{attribute 'TcDependOnClassFactory' := 'Welding_Control_Circle_86s'}
FUNCTION_BLOCK FB_Welding_Control_Circle_86s EXTENDS FB_TcMatSimObject
VAR_INPUT
	stInput: ST_Welding_Control_Circle_86s_Input;
END_VAR
VAR_OUTPUT
	stOutput: ST_Welding_Control_Circle_86s_Output;
END_VAR
VAR
	stInitData: ST_Welding_Control_Circle_86s_InitData;
	arrDataAreas: ARRAY[1..2] OF ST_TcMatSimObjectDataAreaInfo;
	bParametersVerified: BOOL;
END_VAR

PROPERTY CallBy_Online : TctModuleCallByType
GET
hResult := GetObjPara(16#00000000,sizeof(CallBy_Online),adr(CallBy_Online));
END_GET
SET
hResult := SetObjPara(16#00000000,sizeof(CallBy_Online),adr(CallBy_Online));
END_SET
END_PROPERTY

PROPERTY CallBy_Startup : TctModuleCallByType
GET
CallBy_Startup := stInitData.CallBy;
END_GET
SET
stInitData.CallBy := CallBy_Startup;
END_SET
END_PROPERTY

PROPERTY ContextInfoArr_0_TaskCycleTimeNs_Online : UDINT
GET
hResult := GetObjPara(16#03002080,sizeof(ContextInfoArr_0_TaskCycleTimeNs_Online),adr(ContextInfoArr_0_TaskCycleTimeNs_Online));
END_GET
SET
hResult := SetObjPara(16#03002080,sizeof(ContextInfoArr_0_TaskCycleTimeNs_Online),adr(ContextInfoArr_0_TaskCycleTimeNs_Online));
END_SET
END_PROPERTY

PROPERTY ContextInfoArr_0_TaskCycleTimeNs_Startup : UDINT
GET
ContextInfoArr_0_TaskCycleTimeNs_Startup := stInitData.ContextInfoArr_0_TaskCycleTimeNs;
END_GET
SET
stInitData.ContextInfoArr_0_TaskCycleTimeNs := ContextInfoArr_0_TaskCycleTimeNs_Startup;
END_SET
END_PROPERTY

PROPERTY ContextInfoArr_0_TaskOid_Online : OTCID
GET
hResult := GetObjPara(16#03002060,sizeof(ContextInfoArr_0_TaskOid_Online),adr(ContextInfoArr_0_TaskOid_Online));
END_GET
SET
hResult := SetObjPara(16#03002060,sizeof(ContextInfoArr_0_TaskOid_Online),adr(ContextInfoArr_0_TaskOid_Online));
END_SET
END_PROPERTY

PROPERTY ContextInfoArr_0_TaskOid_Startup : OTCID
GET
ContextInfoArr_0_TaskOid_Startup := stInitData.ContextInfoArr_0_TaskOid;
END_GET
SET
stInitData.ContextInfoArr_0_TaskOid := ContextInfoArr_0_TaskOid_Startup;
END_SET
END_PROPERTY

PROPERTY ContextInfoArr_0_TaskPort_Online : UINT
GET
hResult := GetObjPara(16#03002090,sizeof(ContextInfoArr_0_TaskPort_Online),adr(ContextInfoArr_0_TaskPort_Online));
END_GET
SET
hResult := SetObjPara(16#03002090,sizeof(ContextInfoArr_0_TaskPort_Online),adr(ContextInfoArr_0_TaskPort_Online));
END_SET
END_PROPERTY

PROPERTY ContextInfoArr_0_TaskPort_Startup : UINT
GET
ContextInfoArr_0_TaskPort_Startup := stInitData.ContextInfoArr_0_TaskPort;
END_GET
SET
stInitData.ContextInfoArr_0_TaskPort := ContextInfoArr_0_TaskPort_Startup;
END_SET
END_PROPERTY

PROPERTY ContextInfoArr_0_TaskPriority_Online : UDINT
GET
hResult := GetObjPara(16#03002070,sizeof(ContextInfoArr_0_TaskPriority_Online),adr(ContextInfoArr_0_TaskPriority_Online));
END_GET
SET
hResult := SetObjPara(16#03002070,sizeof(ContextInfoArr_0_TaskPriority_Online),adr(ContextInfoArr_0_TaskPriority_Online));
END_SET
END_PROPERTY

PROPERTY ContextInfoArr_0_TaskPriority_Startup : UDINT
GET
ContextInfoArr_0_TaskPriority_Startup := stInitData.ContextInfoArr_0_TaskPriority;
END_GET
SET
stInitData.ContextInfoArr_0_TaskPriority := ContextInfoArr_0_TaskPriority_Startup;
END_SET
END_PROPERTY

PROPERTY ContextInfoArr_0_TaskSortOrder_Online : UDINT
GET
hResult := GetObjPara(16#030020b0,sizeof(ContextInfoArr_0_TaskSortOrder_Online),adr(ContextInfoArr_0_TaskSortOrder_Online));
END_GET
SET
hResult := SetObjPara(16#030020b0,sizeof(ContextInfoArr_0_TaskSortOrder_Online),adr(ContextInfoArr_0_TaskSortOrder_Online));
END_SET
END_PROPERTY

PROPERTY ContextInfoArr_0_TaskSortOrder_Startup : UDINT
GET
ContextInfoArr_0_TaskSortOrder_Startup := stInitData.ContextInfoArr_0_TaskSortOrder;
END_GET
SET
stInitData.ContextInfoArr_0_TaskSortOrder := ContextInfoArr_0_TaskSortOrder_Startup;
END_SET
END_PROPERTY

PROPERTY CycleUpdateExecuted_Online : BOOL
GET
hResult := GetObjPara(16#00000004,sizeof(CycleUpdateExecuted_Online),adr(CycleUpdateExecuted_Online));
END_GET
SET
hResult := SetObjPara(16#00000004,sizeof(CycleUpdateExecuted_Online),adr(CycleUpdateExecuted_Online));
END_SET
END_PROPERTY

METHOD Execute : HRESULT

IF (SUCCEEDED(hResult)) THEN
  hResult := VerifyParameters();
END_IF

	// update DataArea information
SetDataAreaInfo(ADR(arrDataAreas),2);
	
	// call base method
Execute := SUPER^.Execute();
END_METHOD

PROPERTY ExecuteModelCode_Online : BOOL
GET
hResult := GetObjPara(16#00000008,sizeof(ExecuteModelCode_Online),adr(ExecuteModelCode_Online));
END_GET
SET
hResult := SetObjPara(16#00000008,sizeof(ExecuteModelCode_Online),adr(ExecuteModelCode_Online));
END_SET
END_PROPERTY

PROPERTY ExecuteModelCode_Startup : BOOL
GET
ExecuteModelCode_Startup := stInitData.ExecuteModelCode;
END_GET
SET
stInitData.ExecuteModelCode := ExecuteModelCode_Startup;
END_SET
END_PROPERTY

PROPERTY ExecutionSequence_Online : TctModuleExecutionSequenceType
GET
hResult := GetObjPara(16#00000001,sizeof(ExecutionSequence_Online),adr(ExecutionSequence_Online));
END_GET
SET
hResult := SetObjPara(16#00000001,sizeof(ExecutionSequence_Online),adr(ExecutionSequence_Online));
END_SET
END_PROPERTY

PROPERTY ExecutionSequence_Startup : TctModuleExecutionSequenceType
GET
ExecutionSequence_Startup := stInitData.ExecutionSequence;
END_GET
SET
stInitData.ExecutionSequence := ExecutionSequence_Startup;
END_SET
END_PROPERTY

METHOD FB_init : BOOL
VAR_INPUT
	/// if TRUE, the retain variables are initialized (warm start / cold start)
	bInitRetains: BOOL;
	/// if TRUE, the instance afterwards gets moved into the copy code (online change)
	bInCopyCode: BOOL;
	oid: OTCID;
END_VAR
VAR
	clsId: CLSID;
END_VAR

// initialize flags
bParametersVerified := false;
                    
// set module class id for compatibility check
clsId.Data1 := 16#4f7c9520;
clsId.Data2 := 16#5e7b;
clsId.Data3 := 16#4579;
clsId.Data4[0] := 16#be;
clsId.Data4[1] := 16#6e;
clsId.Data4[2] := 16#10;
clsId.Data4[3] := 16#c0;
clsId.Data4[4] := 16#eb;
clsId.Data4[5] := 16#37;
clsId.Data4[6] := 16#31;
clsId.Data4[7] := 16#6d;

AssignClassId(clsId);
                    
// initialize InitData structure with default values              
stInitData.CallByHdr.indexGroup := 0;
stInitData.CallByHdr.indexOffset := 16#00000000;
stInitData.CallByHdr.cbData := SIZEOF(stInitData.CallBy);
stInitData.CallBy := TctModuleCallByType.Module;
stInitData.ExecutionSequenceHdr.indexGroup := 0;
stInitData.ExecutionSequenceHdr.indexOffset := 16#00000001;
stInitData.ExecutionSequenceHdr.cbData := SIZEOF(stInitData.ExecutionSequence);
stInitData.ExecutionSequence := TctModuleExecutionSequenceType.StateUpdateAfterOutputMapping;
stInitData.StepSizeHdr.indexGroup := 0;
stInitData.StepSizeHdr.indexOffset := 16#00000002;
stInitData.StepSizeHdr.cbData := SIZEOF(stInitData.StepSize);
stInitData.StepSize := TctStepSizeType.UseTaskCycleTime;
stInitData.ExecuteModelCodeHdr.indexGroup := 0;
stInitData.ExecuteModelCodeHdr.indexOffset := 16#00000008;
stInitData.ExecuteModelCodeHdr.cbData := SIZEOF(stInitData.ExecuteModelCode);
stInitData.ExecuteModelCode := 1;
stInitData.ContextInfoArr_0_TaskOidHdr.indexGroup := 0;
stInitData.ContextInfoArr_0_TaskOidHdr.indexOffset := 16#03002060;
stInitData.ContextInfoArr_0_TaskOidHdr.cbData := SIZEOF(stInitData.ContextInfoArr_0_TaskOid);
stInitData.ContextInfoArr_0_TaskPriorityHdr.indexGroup := 0;
stInitData.ContextInfoArr_0_TaskPriorityHdr.indexOffset := 16#03002070;
stInitData.ContextInfoArr_0_TaskPriorityHdr.cbData := SIZEOF(stInitData.ContextInfoArr_0_TaskPriority);
stInitData.ContextInfoArr_0_TaskCycleTimeNsHdr.indexGroup := 0;
stInitData.ContextInfoArr_0_TaskCycleTimeNsHdr.indexOffset := 16#03002080;
stInitData.ContextInfoArr_0_TaskCycleTimeNsHdr.cbData := SIZEOF(stInitData.ContextInfoArr_0_TaskCycleTimeNs);
stInitData.ContextInfoArr_0_TaskPortHdr.indexGroup := 0;
stInitData.ContextInfoArr_0_TaskPortHdr.indexOffset := 16#03002090;
stInitData.ContextInfoArr_0_TaskPortHdr.cbData := SIZEOF(stInitData.ContextInfoArr_0_TaskPort);
stInitData.ContextInfoArr_0_TaskSortOrderHdr.indexGroup := 0;
stInitData.ContextInfoArr_0_TaskSortOrderHdr.indexOffset := 16#030020b0;
stInitData.ContextInfoArr_0_TaskSortOrderHdr.cbData := SIZEOF(stInitData.ContextInfoArr_0_TaskSortOrder);
stInitData.Header.cbData := SIZEOF(stInitData)-SIZEOF(stInitData.Header);
stInitData.Header.uiElmCnt := 9;


// set pointer to InitData structure
SetInitDataInfo(ADR(stInitData));

// set DataArea information
SetDataAreaInfo(ADR(arrDataAreas),2);
arrDataAreas[1].nDataAreaId := 0;
arrDataAreas[1].nSize := SIZEOF(stInput);
arrDataAreas[1].pPlcVar := ADR(stInput);
arrDataAreas[1].pModuleProcImg := 0;
arrDataAreas[1].eDataAreaType := E_TcMatSimDataAreaType.InputDst;
arrDataAreas[2].nDataAreaId := 1;
arrDataAreas[2].nSize := SIZEOF(stOutput);
arrDataAreas[2].pPlcVar := ADR(stOutput);
arrDataAreas[2].pModuleProcImg := 0;
arrDataAreas[2].eDataAreaType := E_TcMatSimDataAreaType.OutputSrc;


// initialize basic interface pointers and return
FB_init := SUCCEEDED(Init(oid));
END_METHOD

PROPERTY InitData : ST_Welding_Control_Circle_86s_InitData
GET
InitData := stInitData;
END_GET
SET
stInitData := InitData;
END_SET
END_PROPERTY

PROPERTY Input_Online : ExtU_output_WeldingDiameter10_T
GET
hResult := GetObjPara(16#80000000,sizeof(Input_Online),adr(Input_Online));
END_GET
SET
hResult := SetObjPara(16#80000000,sizeof(Input_Online),adr(Input_Online));
END_SET
END_PROPERTY

{attribute 'object_name' := 'Internal_SetObjState'}
METHOD PROTECTED Internal_SetObjState
VAR_INPUT
	hr: REFERENCE TO HRESULT;
	nextState: TCOM_STATE;
END_VAR

// update pointer to InitData structure
SetInitDataInfo(ADR(stInitData));
// call base method
SUPER^.Internal_SetObjState(hr,nextState);
END_METHOD

PROPERTY MdlInitialized_Online : BOOL
GET
hResult := GetObjPara(16#00000003,sizeof(MdlInitialized_Online),adr(MdlInitialized_Online));
END_GET
SET
hResult := SetObjPara(16#00000003,sizeof(MdlInitialized_Online),adr(MdlInitialized_Online));
END_SET
END_PROPERTY

PROPERTY ModuleBuildInfo_Online : TctModuleBuildInfoType
GET
hResult := GetObjPara(16#00000007,sizeof(ModuleBuildInfo_Online),adr(ModuleBuildInfo_Online));
END_GET
SET
hResult := SetObjPara(16#00000007,sizeof(ModuleBuildInfo_Online),adr(ModuleBuildInfo_Online));
END_SET
END_PROPERTY

PROPERTY ModuleInfo_Online : TctModuleInfoType
GET
hResult := GetObjPara(16#00000006,sizeof(ModuleInfo_Online),adr(ModuleInfo_Online));
END_GET
SET
hResult := SetObjPara(16#00000006,sizeof(ModuleInfo_Online),adr(ModuleInfo_Online));
END_SET
END_PROPERTY

{attribute 'object_name' := 'SaveOnlineParametersForInit'}
METHOD SaveOnlineParametersForInit : HRESULT
VAR
	idx: UINT;
	pInitElemHdr: POINTER TO TComInitDataElmHdr;
	pData: PVOID;
	nData: UDINT;
END_VAR
VAR CONSTANT
	nInitDataAlignment: UDINT := 4;
END_VAR

// update pointer to InitData structure
SetInitDataInfo(ADR(stInitData));
// call base method
SaveOnlineParametersForInit := SUPER^.SaveOnlineParametersForInit();
END_METHOD

PROPERTY SimulinkTime_Online : LREAL
GET
hResult := GetObjPara(16#00000005,sizeof(SimulinkTime_Online),adr(SimulinkTime_Online));
END_GET
SET
hResult := SetObjPara(16#00000005,sizeof(SimulinkTime_Online),adr(SimulinkTime_Online));
END_SET
END_PROPERTY

PROPERTY StepSize_Online : TctStepSizeType
GET
hResult := GetObjPara(16#00000002,sizeof(StepSize_Online),adr(StepSize_Online));
END_GET
SET
hResult := SetObjPara(16#00000002,sizeof(StepSize_Online),adr(StepSize_Online));
END_SET
END_PROPERTY

PROPERTY StepSize_Startup : TctStepSizeType
GET
StepSize_Startup := stInitData.StepSize;
END_GET
SET
stInitData.StepSize := StepSize_Startup;
END_SET
END_PROPERTY

{attribute 'object_name' := 'VerifyParameters'}
METHOD PRIVATE VerifyParameters : HRESULT
VAR
	moduleCallByParam: TctModuleCallByType;
END_VAR

IF (bParametersVerified) THEN
  VerifyParameters := Tc2_System.E_HRESULTAdsErr.HRESULT_ADS_NOERROR;
ELSE
  VerifyParameters := GetObjPara(stInitData.CallByHdr.indexOffset,SIZEOF(moduleCallByParam),ADR(moduleCallByParam));
  
  // check the "CallBy" parameter to be set to "Module"
  IF (SUCCEEDED(VerifyParameters) AND (moduleCallByParam <> TctModuleCallByType.Module)) THEN
      VerifyParameters := Tc2_System.E_HRESULTAdsErr.INVALIDPARM;
  END_IF
  
  // set the parameters verified flag
  bParametersVerified := SUCCEEDED(VerifyParameters);
END_IF
END_METHOD

END_FUNCTION_BLOCK

(* stored: Version 1.1.0.1, ProductVersion 3.1.4020.12
   POU FB_Welding_Control_Circle_86s: Id {24caedbc-12b8-4f64-87d2-ff3d3000a21e}, SpecialFunc None
   Property CallBy_Online: Id {b0ca8028-e351-47bf-bb9b-14d3ef97327c}
   Get Get: Id {6b87a339-992d-4def-9c7c-4f4831e892ca}
   Set Set: Id {2d0296a2-cd98-444d-affd-ad431a74fd96}
   Property CallBy_Startup: Id {75a31c6e-d5d3-4099-89f0-32fa07889e25}
   Get Get: Id {ec503190-93eb-49bb-b560-a131c8b036e6}
   Set Set: Id {3d60197c-94f2-4179-8227-48760ac655d0}
   Property ContextInfoArr_0_TaskCycleTimeNs_Online: Id {26354c8b-d4b8-4947-83ae-12eb5fedcbca}
   Get Get: Id {86cb5be8-a652-4a56-858b-9cd87212b3cf}
   Set Set: Id {eb3801b4-cc63-428e-8bdf-ac4e71ba6d7e}
   Property ContextInfoArr_0_TaskCycleTimeNs_Startup: Id {58e01376-5b55-4777-80d7-e5341e9582e1}
   Get Get: Id {c5ead2be-fe22-456e-b432-875d60b46538}
   Set Set: Id {2de17d08-8ab7-4974-ba1c-bd323d14d281}
   Property ContextInfoArr_0_TaskOid_Online: Id {e03973f3-946d-433a-904d-7fcad3a2d0d5}
   Get Get: Id {9b9341af-c6df-4476-8602-e1233cb1d829}
   Set Set: Id {7de2c92b-d743-46c0-a234-5bf8ddd7b802}
   Property ContextInfoArr_0_TaskOid_Startup: Id {b303394b-30c2-49ac-ab86-f83034190e84}
   Get Get: Id {010efdf1-badb-4483-a762-7d28443de22c}
   Set Set: Id {76a4ab55-bb2b-415d-a651-5074c1a2e273}
   Property ContextInfoArr_0_TaskPort_Online: Id {d5b37149-00a3-4c32-9669-3650dd1b995a}
   Get Get: Id {d9c01139-21ef-413c-8d0a-5c999fd21853}
   Set Set: Id {50163db1-ef91-428f-9cb8-763cd0ffcc9c}
   Property ContextInfoArr_0_TaskPort_Startup: Id {9321b405-c94f-42e1-9e98-18d83d326a18}
   Get Get: Id {1c91222b-bc93-40f2-a135-3d1f9988574a}
   Set Set: Id {60b331ed-26a3-4fd6-8b4a-a29c3fdb5e36}
   Property ContextInfoArr_0_TaskPriority_Online: Id {3a2e1460-98c4-48a4-a507-95a027f4002f}
   Get Get: Id {89d8c549-169a-4231-9b28-bbef071e0f2b}
   Set Set: Id {936db6d6-528f-46d3-b658-1a0d14a21a38}
   Property ContextInfoArr_0_TaskPriority_Startup: Id {94441cdf-d717-431c-b93d-1a527396180f}
   Get Get: Id {ec994f33-70ba-492b-8ca8-aa476597da55}
   Set Set: Id {e5dbe693-9c36-4302-a42b-4c971a83234d}
   Property ContextInfoArr_0_TaskSortOrder_Online: Id {e6f74777-7a1d-40f3-8586-79add9599bbf}
   Get Get: Id {15cf9f80-8c12-4c2a-b07f-db2efd4ea0a7}
   Set Set: Id {a6442160-eb49-4b17-be26-840439b55fc9}
   Property ContextInfoArr_0_TaskSortOrder_Startup: Id {cb07d1a3-9808-4643-9521-2ce5a2c3b04f}
   Get Get: Id {985f8c76-c459-4d29-b91f-b55e5d9f92bc}
   Set Set: Id {aa14aaee-965d-4e77-bdb2-d00398131fe5}
   Property CycleUpdateExecuted_Online: Id {2bae5bad-94b3-4a19-80a1-2dc4abb2799d}
   Get Get: Id {a9eaeb0e-9782-49db-b8f8-d0625427f3a3}
   Set Set: Id {76af491f-a20f-436d-b735-436a66a30d5a}
   Method Execute: Id {0530b76c-bca7-4f73-9698-6dd067a5d327}
   Property ExecuteModelCode_Online: Id {f7fefc4a-023a-48c2-aa03-3dc22508d566}
   Get Get: Id {0633e048-c9d5-44d1-9dd2-046720e3fc42}
   Set Set: Id {1f3dbbd7-d5a3-4c80-bf08-f1cea7862153}
   Property ExecuteModelCode_Startup: Id {69e81b4d-9f9f-498d-8194-b9e49ad21359}
   Get Get: Id {8c5cda7f-d60b-46af-a910-08f8898c18fd}
   Set Set: Id {b357b3e1-cf83-4cab-a038-058f2f4623ed}
   Property ExecutionSequence_Online: Id {d861df67-52f3-485e-a024-5600edc355e2}
   Get Get: Id {8f29a9f2-5c97-4244-a6d5-fd1cc066db4a}
   Set Set: Id {e331af35-a644-474a-8257-86cf2c147545}
   Property ExecutionSequence_Startup: Id {ae6c0ac3-2b57-4143-a852-2557b0c0add4}
   Get Get: Id {14d5bc24-8704-4d52-8022-f8f7a0051b06}
   Set Set: Id {85536940-6b79-4d7f-8c00-cacc16e749df}
   Method FB_init: Id {435217ff-0b69-4c3a-9d7d-844bc7a11af9}
   Property InitData: Id {9398d2f8-0fb4-4173-86e1-b77caba42dfc}
   Get Get: Id {63980dce-5e23-40d9-9648-e396ef819cd5}
   Set Set: Id {489bd351-a501-44d5-861b-2a3b0cd37e8c}
   Property Input_Online: Id {5930cb1c-4e8e-4b3b-8810-d262438c0ce2}
   Get Get: Id {67864276-a53e-4d06-a444-033acd93463c}
   Set Set: Id {1953a2f3-fa23-4b3b-8b2f-20fb6c75760a}
   Method Internal_SetObjState: Id {f917191b-bc39-4e93-97dd-82ea91e4972c}
   Property MdlInitialized_Online: Id {297ad590-ce0a-4d4f-ba4b-126724e9f3e4}
   Get Get: Id {d9be9f5a-f6c4-4d6c-a7ec-191150450978}
   Set Set: Id {1c90bd08-f1a1-4d1b-b93f-3e7a3effc85f}
   Property ModuleBuildInfo_Online: Id {c8da72ea-fd68-42e0-8f4a-4e48a3213be6}
   Get Get: Id {a6d789a8-ff0a-483e-ba3f-3a34ea9e3312}
   Set Set: Id {1f1e527a-74d3-4b4f-9404-835fd09a9776}
   Property ModuleInfo_Online: Id {1cda82e7-66f4-4c02-924c-d0d15696bdfe}
   Get Get: Id {48815289-950e-4e90-a853-c2e5787586db}
   Set Set: Id {9c110b75-3c1c-4f17-b830-b9fa90715735}
   Method SaveOnlineParametersForInit: Id {56ccbfde-ad5c-430f-95ec-cbab83084034}
   Property SimulinkTime_Online: Id {a0ee90e1-1c74-45f7-8ff6-a3e5709acdc5}
   Get Get: Id {8eec9dac-7128-4cee-9d44-55428d342fc0}
   Set Set: Id {8ad83c1d-22a8-4e09-b3e4-df0fc330a7b7}
   Property StepSize_Online: Id {446c9e7b-cb1f-457b-bc21-8e4189711aa9}
   Get Get: Id {ee1e590a-2d02-4ce3-8e81-34c39b0fa417}
   Set Set: Id {aab00895-47b1-4a9a-9bda-780a4c8260af}
   Property StepSize_Startup: Id {b002c1ca-5d8e-4cd4-99a9-89665ed9f32c}
   Get Get: Id {aa87d388-bce6-42f0-921b-ec9660d968f0}
   Set Set: Id {2040f6c9-59a3-4c3c-87c3-d41b3fe598dc}
   Method VerifyParameters: Id {db83779f-11a7-40fe-bdaa-cc9ce58e8c11} *)
